Staubli VAL3: onF2Event.pgx

program onF2Event()
begin
  // look if the bButton is enable
  if bButton[1]
    //
  endIf
end
